FUNCTION_BLOCK FB_Smart
VAR_INPUT
END_VAR
VAR_OUTPUT
END_VAR
VAR
END_VAR

END_FUNCTION_BLOCK

(* stored: Version 1.1.0.1
   POU FB_Smart: Id {aac2b053-c49f-4ea3-b34f-53f530ed70d8}, SpecialFunc None *)
